// TIA Portal V20 export
DATA_BLOCK "DB_IO_Config"   // DB810
TITLE = DB_IO_Config
{ S7_Optimized_Access := 'FALSE' }
VERSION : 0.1
// IO test config DB810 non-optimized
// stored: AutoNumber false, IsOnlyStoredInLoadMemory false, IsWriteProtectedInAS false
   VAR
      DI : Array[1..20] of "UDT_DigSlot";
      DQ : Array[1..20] of "UDT_DigSlot";
      AI : Array[1..20] of "UDT_AnaSlot";
      AQ : Array[1..20] of "UDT_AnaSlot";
   END_VAR
BEGIN
END_DATA_BLOCK
